FUNCTION_BLOCK RunETest EXTENDS RunAxisInspection
VAR
	
	//Cylinders
	connectorHolder : POINTER TO RunCylinder;
	cableHolder : POINTER TO RunCylinder;
	plugin : POINTER TO RunCylinder;
	//Sensors
	tongueExistedA : POINTER TO RunSignal;
	tongueExistedB : POINTER TO RunSignal;
	tongueGlueA : POINTER TO RunSignal;
	tongueGlueB : POINTER TO RunSignal;
	//from tester
	ioBundle : POINTER TO ioBundleET;
	//
	isOK : BOOL;
	isRedo : BOOL;
	etSeriesNgCounter : UINT;
	etRedoCounter : UINT;
	//
	block : MaterialBlock;
END_VAR
VAR PERSISTENT
	indexCommandPick : INT := 1;
	indexReleaseConnectorHolder : INT := 1;
	
	etUsageCounter : UINT;
	etUsageThreshold : UINT;
	
	etNgAlarmSwitch : BOOL;
	etSeriesNgThreshold : UINT;
	etRedoGoal : UINT;
END_VAR

SUPER^();

IF etUsageCounter>=etUsageThreshold THEN
	//!Clear by manual operation
	AlarmCode := eErrorCodes.AC_ET_USAGE_MEET; 
END_IF

CASE outputState OF
	eSpecialStates.SLAVE_ENTER_PROCEDURE:
		bSerialTransition := connectorHolder^.Execute(eCylinderCommands.COMMAND_B);
	16#201:
		bSerialTransition := plugin^.Execute(eCylinderCommands.COMMAND_B);
		IF bSerialTransition THEN
			//usage count-up
			etUsageCounter := etUsageCounter+1;
		END_IF
	16#202:
		bSerialTransition := axis1^.ExecuteParameterIndex(indexCommandPick); //down to pick
	16#203:
		bSerialTransition := cableHolder^.Execute(eCylinderCommands.COMMAND_B) ;//hold 
	16#204:
		IF TRUE THEN
			//going to swing
			NextState := eSpecialStates.SLAVE_AXIS_INSPECTION_ENTER;
		END_IF
	//-----------------
	eSpecialStates.SLAVE_AXIS_INSPECTION_EXIT:
		//TODO , read status and report
		isOK := tongueExistedA^.debouncedOn AND tongueExistedB^.debouncedOn AND  tongueGlueA^.debouncedOff AND tongueGlueB^.debouncedOff AND ioBundle^.o3;
		
		isRedo := FALSE;//reset
		IF isOK THEN
			//ok
			etSeriesNgCounter := 0;
		ELSE
			//ng
			etSeriesNgCounter := etSeriesNgCounter+1;
			IF 	(etSeriesNgCounter >= etSeriesNgThreshold) AND etNgAlarmSwitch AND (etRedoCounter >=etRedoGoal) THEN
				//raise alarm
				AlarmCode := eErrorCodes.AC_ET_SERIES_NG;
				etSeriesNgCounter := 0;
			ELSIF etRedoCounter < etRedoGoal THEN
				//not reach , redo
				isRedo := TRUE;
			END_IF
		END_IF		
		//report
		block.data[0] := TO_WORD(isOK);
		block.data[1] := TO_WORD(ioBundle^.o3); //et
		block.data[2] := TO_WORD(tongueExistedA^.debouncedOn);
		block.data[3] := TO_WORD(tongueExistedB^.debouncedOn);
		block.data[4] := TO_WORD(tongueGlueA^.debouncedOff);
		block.data[5] := TO_WORD(tongueGlueB^.debouncedOff);
		SlotBase^.Data := block;
		SlotBase^.Act := TRUE;
		
		bSerialTransition := TRUE;
	16#401:
		bSerialTransition := axis1^.ExecuteParameterIndex(indexCommandPick); //back to to pick
	16#402:
		bSerialTransition := cableHolder^.Execute(eCylinderCommands.COMMAND_A);
	16#403:
		bSerialTransition := plugin^.Execute(eCylinderCommands.COMMAND_A);
	16#404:
		bSerialTransition := connectorHolder^.Execute(eCylinderCommands.COMMAND_A);
	16#405:
		//all axis backto standby
		IF NOT transitionByte.0 AND_THEN axis1^.ExecuteParameterIndex(indexStandByAxis1) THEN
			transitionByte.0 := TRUE;
		END_IF
		IF NOT transitionByte.1 AND_THEN axis2^.ExecuteParameterIndex(indexStandByAxis2) THEN
			transitionByte.1 := TRUE;
		END_IF
		IF transitionByte=3 THEN
			IF isRedo THEN
				etRedoCounter := etRedoCounter+1;
				NextState := eSpecialStates.SLAVE_ENTER_PROCEDURE;
			ELSE
				etRedoCounter :=0; //reset
				NextState := eSpecialStates.SLAVE_WORK_DONE;
			END_IF
		END_IF
END_CASE
//release to swing // release connector holder when horizon moving
IF (slaveWorkingSignal[1] AND ((nCounter=indexReleaseConnectorHolder AND_THEN connectorHolder^.Execute(eCylinderCommands.COMMAND_A)) OR nCounter<>indexReleaseConnectorHolder)) THEN
	slaveWorkingSignal[1] := FALSE;
END_IF

METHOD FB_init : BOOL
VAR_INPUT
	bInitRetains : BOOL; // if TRUE, the retain variables are initialized (warm start / cold start)
	bInCopyCode : BOOL;  // if TRUE, the instance afterwards gets moved into the copy code (online change)
	
	argParent : POINTER TO RunUnitGeneric;
	argSlotBase : POINTER TO RunMaterial;
	argSlotLast : POINTER TO RunMaterial;
	
	argWorkingSignal : POINTER TO BOOL;
	
	argAxis1 : POINTER TO RunAxis;
	argAxis2 : POINTER TO RunAxis;
	
	argSideAligner : pointer to RunCylinder;
	
	argConnectorHolder : POINTER TO RunCylinder;
	argCableHolder : POINTER TO RunCylinder;
	argPlugin : POINTER TO RunCylinder;
	//Sensors
	argTongueExistedA : POINTER TO RunSignal;
	argTongueExistedB : POINTER TO RunSignal;
	argTongueGlueA : POINTER TO RunSignal;
	argTongueGlueB : POINTER TO RunSignal;
	
	argIoBundle : pointer to ioBundleET;
END_VAR
//initialize 
Parent := argParent;
SlotBase := argSlotBase;
SlotLast := argSlotLast;
//
IF bInitRetains THEN
	NextState := eSpecialStates.INITIAL_BEGIN;
END_IF

workingSignal := argWorkingSignal; //link

axis1 := argAxis1;
axis2 := argAxis2;

//
connectorHolder := argConnectorHolder;
cableHolder :=argCableHolder;
plugin :=argPlugin;
	//Sensors
tongueExistedA :=argTongueExistedA;
tongueExistedB :=argTongueExistedB;
tongueGlueA :=argTongueGlueA;
tongueGlueB :=argTongueGlueB;
ioBundle := argIoBundle;
END_METHOD

METHOD Initialize : BOOL
VAR_INPUT
END_VAR

CASE outputState OF
	eSpecialStates.INITIAL_BEGIN:
		// release all cylinder
		IF NOT transitionByte.0 AND_THEN plugin^.Execute(argCommand:= eCylinderCommands.COMMAND_A) THEN
			transitionByte.0 := TRUE;
		END_IF
		IF NOT transitionByte.1 AND_THEN connectorHolder^.Execute(argCommand:= eCylinderCommands.COMMAND_A) THEN
			transitionByte.1 := TRUE;
		END_IF
		IF NOT transitionByte.2 AND_THEN cableHolder^.Execute(argCommand:= eCylinderCommands.COMMAND_A) THEN
			transitionByte.2 := TRUE;
		END_IF
		IF transitionByte=7 THEN
			NextState := eSpecialStates.INITIAL_STATE_7; // to return axis
		END_IF
END_CASE


Initialize:= SUPER^.Initialize(); //do axis return
END_METHOD

END_FUNCTION_BLOCK

(* stored: Version 1.1.0.1, ProductVersion 3.1.4022.10
   POU RunETest: Id {72e72744-8d8b-4127-a1f7-17ac70d49060}, SpecialFunc None
   Method FB_init: Id {efefce5e-b774-42d4-a90d-6714e5f02940}
   Method Initialize: Id {b1cb528c-756c-4543-b261-8a9a85e25c02} *)
